PROGRAM MAIN
VAR
END_VAR

END_PROGRAM

(* stored: Version 1.1.0.1
   POU MAIN: Id {0de7b7dd-5ad8-47ee-97be-c32642f4f628} *)
